Yaskawa INFORM job: OK_R2_O24B(90,0)KMOK.JBI

/JOB
//NAME OK_R2_O24B(90,0)KMOK
///FOLDERNAME X4
//POS
///NPOS 232,232,232,13,0,0
///TOOL 0
///POSTYPE PULSE
///PULSE
C00000=-110421,-114568,-128442,-17543,109310,40994
C00001=-110421,-114568,-128442,-17543,109310,40994
C00002=-114535,-118016,-126260,-17193,105500,40103
C00003=-116189,-118926,-125238,-17079,104117,39719
C00004=-122470,-118801,-125267,-16970,102934,37675
C00005=-122542,-119768,-123081,-16831,101153,37902
C00006=-122470,-118801,-125267,-16970,102934,37675
C00007=-116189,-118926,-125238,-17079,104117,39719
C00008=-115768,-121709,-122546,-16840,101244,40278
C00009=-119833,-121860,-122638,-16796,100405,38960
C00010=-115768,-121709,-122546,-16840,101244,40278
C00011=-116189,-118926,-125238,-17079,104117,39719
C00012=-114535,-118016,-126260,-17193,105500,40103
C00013=-110421,-114568,-128442,-17543,109310,40994
C00014=-126378,-115954,-129597,15290,109099,-41008
C00015=-122420,-119367,-127301,14983,105339,-40105
C00016=-120830,-120251,-126232,14883,103983,-39719
C00017=-114862,-120096,-125989,14784,102865,-37775
C00018=-115075,-121077,-123808,14669,101114,-38064
C00019=-114862,-120096,-125989,14784,102865,-37775
C00020=-120830,-120251,-126232,14883,103983,-39719
C00021=-121393,-120121,-122865,14745,102140,-40145
C00022=-117360,-120220,-122765,14697,101321,-38836
C00023=-121393,-120121,-122865,14745,102140,-40145
C00024=-120830,-120251,-126232,14883,103983,-39719
C00025=-122420,-119367,-127301,14983,105339,-40105
C00026=-126378,-115954,-129597,15290,109099,-41008
C00027=-68546,-106272,-120466,15386,126682,-61056
C00028=-65872,-117617,-121364,15125,121103,-60799
C00029=-65994,-124789,-121483,14506,117628,-61338
C00030=-65994,-124776,-119887,14364,116682,-61464
C00031=-64727,-121841,-121551,15095,118908,-60654
C00032=-66354,-118147,-119193,14717,119632,-61205
C00033=-63947,-125385,-121489,15018,116968,-60618
C00034=-66354,-118147,-119193,14717,119632,-61205
C00035=-67446,-114060,-119015,14744,121753,-61346
C00036=-69995,-103128,-118158,14981,127125,-61604
C00037=-43458,-109907,-123851,22079,119459,-51827
C00038=-39582,-118676,-123782,21672,114241,-51374
C00039=-37960,-121735,-123576,21587,112243,-51139
C00040=-38039,-122241,-121246,21299,110682,-51473
C00041=-37960,-121735,-123576,21587,112243,-51139
C00042=-39439,-119560,-121458,21353,112446,-51673
C00043=-35892,-124835,-123088,21550,109947,-50789
C00044=-39439,-119560,-121458,21353,112446,-51673
C00045=-41022,-116597,-121679,21425,114395,-51908
C00046=-44803,-108153,-121807,21787,119465,-52368
C00047=-46269,-104607,-116900,14890,131588,-81597
C00048=-45575,-117487,-118566,13929,126044,-82146
C00049=-45272,-122474,-119074,13631,123805,-82329
C00050=-45097,-121786,-116375,13476,122503,-82429
C00051=-45272,-122474,-119074,13631,123805,-82329
C00052=-54794,-132635,-122270,15461,117667,-84057
C00053=-51488,-139835,-124335,16145,114686,-83176
C00054=-54794,-132635,-122270,15461,117667,-84057
C00055=-54354,-108181,-111858,18613,130239,-82011
C00056=-56948,-114588,-113873,16794,128830,-83498
C00057=-54354,-108181,-111858,18613,130239,-82011
C00058=-54354,-108181,-111858,18613,105079,-82011
C00059=-125473,-127815,-125744,-20402,114696,66128
C00060=-144354,-128645,-122856,-20089,112993,66444
C00061=-144356,-128558,-121667,-19978,112345,66561
C00062=-143692,-123642,-120175,-20108,114021,66516
C00063=-144449,-128577,-122916,-20120,113038,66399
C00064=-144368,-128510,-121483,-19685,112887,66475
C00065=-144076,-129076,-121363,-22700,108650,60338
C00066=-144065,-129172,-121967,-22849,108765,60054
C00067=-145562,-127750,-121174,10660,122518,78224
C00068=-145562,-127687,-120572,10615,122186,78189
C00069=-144870,-122921,-119115,11103,123620,78631
C00070=-145668,-127710,-121822,10673,122944,78224
C00071=-145551,-127683,-120865,10446,122273,78190
C00072=-145550,-127738,-121466,10490,122609,78224
C00073=-145528,-127702,-122047,10145,122795,78223
C00074=-145466,-127681,-122511,8080,122804,78067
C00075=-145466,-127654,-121910,8044,122451,78039
C00076=-144776,-122735,-120395,8485,123961,78447
C00077=-145489,-127675,-123160,8112,123205,78089
C00078=-145462,-127615,-121976,8108,122518,78051
C00079=-145461,-127639,-122576,8144,122872,78079
C00080=-145470,-127509,-122616,9202,123100,78187
C00081=-145470,-127489,-122014,9161,122745,78155
C00082=-144781,-122556,-120500,9628,124248,78581
C00083=-145526,-127464,-123250,9229,123515,78201
C00084=-145457,-127452,-122138,8905,122802,78142
C00085=-145457,-127468,-122738,8946,123159,78173
C00086=-145419,-127422,-123013,7792,123191,78085
C00087=-145369,-127281,-122655,6352,123642,78005
C00088=-145369,-127269,-122086,6324,123301,77983
C00089=-144684,-122332,-120516,6740,124807,78367
C00090=-145346,-127303,-123341,6395,124049,78040
C00091=-145359,-127218,-122002,6175,123337,77977
C00092=-145359,-127231,-122569,6203,123677,77998
C00093=-145369,-127141,-122578,7278,123283,78064
C00094=-145369,-127129,-121996,7245,122933,78039
C00095=-144683,-122199,-120454,7674,124442,78435
C00096=-145369,-127140,-123243,7317,123689,78093
C00097=-145374,-127101,-121995,7642,122781,78062
C00098=-145373,-127113,-122583,7677,123134,78088
C00099=-145323,-127035,-122273,5816,123755,77984
C00100=-145301,-126904,-121478,4974,124764,77984
C00101=-145245,-126972,-122476,3510,122733,77759
C00102=-145245,-126962,-121900,3495,122385,77747
C00103=-144566,-122041,-120337,3835,123918,78081
C00104=-145130,-127078,-123177,3572,123105,77819
C00105=-145235,-126936,-121864,3341,122099,77723
C00106=-145235,-126947,-122445,3356,122451,77734
C00107=-145235,-126704,-121159,4007,122972,77833
C00108=-145235,-126667,-120590,3990,122642,77820
C00109=-144560,-121896,-119039,4346,124100,78159
C00110=-145144,-126819,-121880,4063,123351,77885
C00111=-145222,-126734,-121009,3552,122070,77754
C00112=-143543,-128240,-121764,3717,120897,78337
C00113=-144110,-127812,-122791,3542,121772,78139
C00114=-145205,-126597,-125313,3216,123991,77765
C00115=-78497,-119087,-126940,-8466,133839,13526
C00116=-78488,-120793,-123596,-8031,130934,13800
C00117=-78485,-121192,-122172,-7887,129863,13894
C00118=-78455,-120845,-123307,-7986,130735,13833
C00119=-77443,-125885,-123641,-7190,128464,14473
C00120=-78479,-121212,-122221,-7886,129884,13896
C00121=-78482,-120810,-123644,-8031,130956,13801
C00122=-78491,-119095,-126985,-8467,133863,13526
C00123=-78416,-117369,-129459,12992,98157,11559
C00124=-78415,-119818,-126610,12888,95218,11250
C00125=-78415,-120492,-125378,12858,94139,11138
C00126=-77369,-125600,-126977,12690,92378,11308
C00127=-78323,-119762,-126393,12873,95102,11269
C00128=-78420,-120510,-125276,12857,94070,11129
C00129=-78420,-119847,-126511,12886,95145,11241
C00130=-78422,-117430,-129370,12989,98073,11548
C00131=-84214,-85469,-118328,4842,91147,7442
C00132=-74059,-12147,-76922,1404,102997,10572
C00133=-133925,-71820,-61688,-34619,64887,29675
C00134=-146663,-27707,-36323,-28508,66625,23960
C00135=-151246,10085,-12654,-25869,69264,21358
C00136=-177412,39753,198,-10194,88087,11090
C00137=-178299,46865,9603,8268,86130,11567
C00138=-176438,52797,17986,7782,83863,12031
C00139=-176438,52484,19424,7790,82827,11968
C00140=-176438,52797,17986,7782,83863,12031
C00141=-176227,55662,21169,7731,83361,12069
C00142=-176438,52797,17986,7782,83863,12031
C00143=-178195,43565,7177,-9991,85692,11029
C00144=-179304,50598,16552,-9714,83440,10842
C00145=-179945,54564,20926,-9550,82718,10686
C00146=-179817,54163,20479,-9581,82800,10721
C00147=-179817,53892,21980,-9596,81755,10803
C00148=-179304,50598,16552,-9714,83440,10842
C00149=-179304,50598,16552,-9714,83440,10842
C00150=-178927,45721,9401,-9794,85349,10816
C00151=-178167,41839,2311,-9989,87773,10872
C00152=-183075,42459,3197,-17469,92450,20343
C00153=-184391,45146,9017,-17153,90080,20237
C00154=-187277,51257,17514,-16512,87509,19616
C00155=-187277,51016,18753,-16517,86658,19730
C00156=-187277,51257,17514,-16512,87509,19616
C00157=-187989,53981,20519,-16358,86938,19449
C00158=-187277,51257,17514,-16512,87509,19616
C00159=-185546,45393,8874,-16907,90057,19851
C00160=-188954,54144,18535,-20814,94698,27736
C00161=-189948,54829,23502,-24427,90749,27662
C00162=-189948,54721,24380,-24417,90207,27773
C00163=-189948,54829,23502,-24427,90749,27662
C00164=-190693,55997,24806,-24308,90350,27474
C00165=-189948,54829,23502,-24427,90749,27662
C00166=-191226,46719,10370,-23503,99774,32576
C00167=-194241,47366,13370,-23088,97565,31938
C00168=-194241,47163,14282,-23044,96951,32058
C00169=-194241,47366,13370,-23088,97565,31938
C00170=-195479,48868,14996,-22944,97022,31602
C00171=-194241,47366,13370,-23088,97565,31938
C00172=-191615,46469,10340,-23456,99568,32478
C00173=-181855,44977,8339,-27183,101400,42897
C00174=-186261,52191,18476,-27626,103380,47450
C00175=-186261,52000,19461,-27536,102751,47603
C00176=-186261,52191,18476,-27626,103380,47450
C00177=-187017,51834,18080,-27612,103190,47211
C00178=-186261,52191,18476,-27626,103380,47450
C00179=-171257,48190,12361,-32854,103470,53443
C00180=-172498,42405,8067,-32730,102732,53174
C00181=-172498,42136,9154,-32614,102046,53379
C00182=-172498,42405,8067,-32730,102732,53174
C00183=-173166,39976,5518,-32734,102755,52903
C00184=-172498,42405,8067,-32730,102732,53174
C00185=-171464,48985,12939,-32850,103438,53371
C00186=-169687,51444,12946,-33160,105162,53551
C00187=-184933,42158,3162,-30363,102223,10869
C00188=-186478,44106,8144,-29956,99900,10911
C00189=-188964,49864,16491,-29066,96066,9719
C00190=-187085,45252,9276,-29882,99600,10761
C00191=-186375,44289,9504,-29889,99288,11112
C00192=-188932,49894,16522,-29069,96073,9729
C00193=-187598,64926,30953,-23001,93658,11625
C00194=-184091,69419,36163,-18103,87388,9711
C00195=-183329,49111,13525,-21934,85838,-1831
C00196=-182560,45031,6210,-22112,88271,-2010
C00197=-164611,45054,6259,-27542,116257,62631
C00198=-165962,40795,4672,-27363,114755,62481
C00199=-168804,37690,3528,-27392,113071,61778
C00200=-167727,42077,8101,-27182,112908,62250
C00201=-168804,38233,1799,-27701,114270,61464
C00202=-172036,45397,11586,-27411,111162,60980
C00203=-173961,50198,16751,-27391,109920,60533
C00204=-173988,50269,16828,-27390,109902,60527
C00205=-175518,40442,6505,-27349,101254,50892
C00206=-176418,41479,8497,-27978,96504,46634
C00207=-174286,53569,18433,-27340,100959,51234
C00208=-172614,55478,17651,-27620,102791,51416
C00209=-179054,42000,3002,-22996,89562,-1047
C00210=-179906,45884,10050,-22784,87172,-886
C00211=-179980,55307,22142,-22805,84750,-451
C00212=-180237,47802,12025,-22705,86872,-945
C00213=-179743,45860,11189,-22831,86556,-712
C00214=-179765,55798,22804,-22861,84662,-356
C00215=-179423,51484,18060,-14503,78815,-9583
C00216=-178933,49946,16450,-4188,75758,-19147
C00217=-177518,54886,19966,-905,79614,-18236
C00218=-175510,52869,17962,2143,79991,-17090
C00219=-179383,44561,8630,-4008,77771,-19367
C00220=-179878,42216,-2358,-3772,83293,-19698
C00221=-181279,19301,-18084,-30673,107641,36259
C00222=-186954,17040,-16309,-29931,103762,35153
C00223=-186474,43263,7155,-30055,116560,25020
C00224=-185760,43661,8832,-29744,116081,25463
C00225=-186986,17160,-16198,-29927,103745,35146
C00226=-192293,22649,-14002,-21464,99552,35428
C00227=-191916,35450,-1506,-21432,98603,35730
C00228=-192278,42179,5472,-18084,93007,29470
C00229=-192157,46216,9774,-15899,90290,26168
C00230=-185951,26886,-15636,-17349,96949,27318
C00231=-180469,24600,-14591,-31088,105394,11680
BC00000=365735,697660,1075175
BC00001=365735,826919,1075175
BC00002=365735,826919,1075175
BC00003=365735,826919,1075175
BC00004=365735,826919,1075175
BC00005=365735,826919,1075175
BC00006=365735,826919,1075175
BC00007=365735,826919,1075175
BC00008=365735,826919,1075175
BC00009=365735,826919,1075175
BC00010=365735,826919,1075175
BC00011=365735,826919,1075175
BC00012=365735,826919,1075175
BC00013=365735,826919,1075175
BC00014=303667,828438,1075175
BC00015=303667,828438,1075175
BC00016=303667,828438,1075175
BC00017=303667,828438,1075175
BC00018=303667,828438,1075175
BC00019=303667,828438,1075175
BC00020=303667,828438,1075175
BC00021=303667,828438,1075175
BC00022=303667,828438,1075175
BC00023=303667,828438,1075175
BC00024=303667,828438,1075175
BC00025=303667,828438,1075175
BC00026=303667,828438,1075175
BC00027=337741,890424,1075175
BC00028=337741,890424,1075175
BC00029=337741,890424,1075175
BC00030=337741,890424,1075175
BC00031=337741,890424,1075175
BC00032=337741,890424,1075175
BC00033=337741,890424,1075175
BC00034=337741,890424,1075175
BC00035=337741,890424,1075175
BC00036=337741,890424,1075175
BC00037=224426,912763,1075175
BC00038=224426,912763,1075175
BC00039=224426,912763,1075175
BC00040=224426,912763,1075175
BC00041=224426,912763,1075175
BC00042=224426,912763,1075175
BC00043=224426,912763,1075175
BC00044=224426,912763,1075175
BC00045=224426,912763,1075175
BC00046=224426,912763,1075175
BC00047=171301,903205,1075175
BC00048=171301,903205,1075175
BC00049=171301,903205,1075175
BC00050=171301,903205,1075175
BC00051=171301,903205,1075175
BC00052=171301,903205,1075175
BC00053=171301,903205,1075175
BC00054=171301,903205,1075175
BC00055=171301,903205,1075175
BC00056=171301,903205,1075175
BC00057=171301,903205,1075175
BC00058=171301,903205,1075175
BC00059=269606,880492,1075175
BC00060=267821,875290,1075175
BC00061=267108,873210,1075175
BC00062=267108,873210,1075175
BC00063=267108,873210,1075175
BC00064=264556,874058,1075175
BC00065=269924,868703,1075175
BC00066=270646,869481,1075175
BC00067=229357,874448,1075175
BC00068=229412,873357,1075175
BC00069=229412,873357,1075175
BC00070=229412,873357,1075175
BC00071=236091,873318,1075175
BC00072=236043,874407,1075175
BC00073=249309,874312,1075175
BC00074=258931,874853,1075175
BC00075=258932,873778,1075175
BC00076=258932,873778,1075175
BC00077=258932,873778,1075175
BC00078=265217,873784,1075175
BC00079=265214,874859,1075175
BC00080=282651,874653,1075175
BC00081=282689,873584,1075175
BC00082=282689,873584,1075175
BC00083=282689,873584,1075175
BC00084=289464,873670,1075175
BC00085=289435,874740,1075175
BC00086=298152,875065,1075175
BC00087=312070,876808,1075175
BC00088=312063,875684,1075175
BC00089=312063,875684,1075175
BC00090=312063,875684,1075175
BC00091=318618,875875,1075175
BC00092=318629,877004,1075175
BC00093=336326,875802,1075175
BC00094=336344,874702,1075175
BC00095=336344,874702,1075175
BC00096=336344,874702,1075175
BC00097=342221,874261,1075175
BC00098=342191,875351,1075175
BC00099=344956,877512,1075175
BC00100=345746,880197,1075175
BC00101=367558,876774,1075175
BC00102=367507,875664,1075175
BC00103=367507,875664,1075175
BC00104=367507,875664,1075175
BC00105=374249,875310,1075175
BC00106=374309,876411,1075175
BC00107=391669,878109,1075175
BC00108=391646,876972,1075175
BC00109=391646,876972,1075175
BC00110=391646,876972,1075175
BC00111=394320,875907,1075175
BC00112=398174,874845,1075175
BC00113=398174,876946,1075175
BC00114=397796,882197,1075175
BC00115=322205,870699,1075175
BC00116=319350,870698,1075175
BC00117=318208,870697,1075175
BC00118=318208,870697,1075175
BC00119=318208,870697,1075175
BC00120=313667,870683,1075175
BC00121=314809,870684,1075175
BC00122=317664,870685,1075175
BC00123=260517,820620,1075175
BC00124=262870,823684,1075175
BC00125=263812,824910,1075175
BC00126=263812,824910,1075175
BC00127=263812,824910,1075175
BC00128=267687,824922,1075175
BC00129=266745,823696,1075175
BC00130=264392,820632,1075175
BC00131=264392,769677,1075175
BC00132=221812,674137,1075175
BC00133=202699,680494,271587
BC00134=202699,714122,185597
BC00135=202699,732276,139175
BC00136=202699,826035,116002
BC00137=202699,826035,116002
BC00138=202699,826035,116002
BC00139=202699,826035,116002
BC00140=202699,826035,116002
BC00141=202699,826035,116002
BC00142=202699,826035,116002
BC00143=202699,826035,116002
BC00144=202699,826035,116002
BC00145=202699,826035,116002
BC00146=202699,826035,116002
BC00147=202699,826035,116002
BC00148=202699,826035,116002
BC00149=202699,826035,116002
BC00150=202699,826035,116002
BC00151=202699,826035,116002
BC00152=214146,822500,117016
BC00153=214146,822500,117016
BC00154=214146,822501,117010
BC00155=214146,822501,117010
BC00156=214146,822501,117010
BC00157=214146,822501,117010
BC00158=214146,822501,117010
BC00159=214146,822500,117016
BC00160=227542,823667,115727
BC00161=227542,823667,115727
BC00162=227542,823667,115727
BC00163=227542,823667,115727
BC00164=227542,823667,115727
BC00165=227542,823667,115727
BC00166=236387,824437,114876
BC00167=236387,824436,114874
BC00168=236387,824436,114874
BC00169=236387,824436,114874
BC00170=236387,824436,114874
BC00171=236387,824436,114874
BC00172=236387,824437,114876
BC00173=241078,796619,103509
BC00174=241078,796619,103509
BC00175=241078,796619,103509
BC00176=241078,796619,103509
BC00177=241078,796619,103509
BC00178=241078,796619,103509
BC00179=245862,768255,91919
BC00180=245862,768255,91917
BC00181=245862,768255,91917
BC00182=245862,768255,91917
BC00183=245862,768255,91917
BC00184=245862,768255,91917
BC00185=245862,768255,91919
BC00186=245862,768255,91919
BC00187=217247,830516,95414
BC00188=217247,830516,95414
BC00189=217248,830516,95407
BC00190=217247,830516,95414
BC00191=217247,830516,95414
BC00192=217248,830516,95407
BC00193=217248,830516,95411
BC00194=217248,830516,95408
BC00195=217247,830516,95414
BC00196=217247,830516,95414
BC00197=224251,767755,101593
BC00198=224251,767755,101593
BC00199=224251,767755,101593
BC00200=224251,767755,101593
BC00201=224251,767755,101593
BC00202=224251,767755,101593
BC00203=224251,767755,101593
BC00204=224251,767755,101593
BC00205=224251,767755,101593
BC00206=224251,767755,101593
BC00207=224251,767755,101593
BC00208=224251,767755,101593
BC00209=207177,824936,95452
BC00210=207177,824936,95452
BC00211=207177,824936,95452
BC00212=207177,824936,95452
BC00213=207177,824936,95452
BC00214=207177,824936,95452
BC00215=207177,824936,95452
BC00216=207178,824936,95451
BC00217=207178,824936,95451
BC00218=207178,824936,95451
BC00219=207177,824936,95452
BC00220=207177,824936,95452
BC00221=219397,819007,95367
BC00222=219397,819007,95367
BC00223=219398,819006,95372
BC00224=219398,819006,95372
BC00225=219397,819007,95367
BC00226=219397,819007,95367
BC00227=219397,819007,95367
BC00228=219397,819007,95367
BC00229=219397,819007,95367
BC00230=219397,819007,95367
BC00231=219398,819006,95372
EC00000=798156,0
EC00001=798156,0
EC00002=798156,0
EC00003=798156,0
EC00004=798156,0
EC00005=798156,0
EC00006=798156,0
EC00007=798156,0
EC00008=798156,0
EC00009=798156,0
EC00010=798156,0
EC00011=798156,0
EC00012=798156,0
EC00013=798156,0
EC00014=798156,0
EC00015=798156,0
EC00016=798156,0
EC00017=798156,0
EC00018=798156,0
EC00019=798156,0
EC00020=798156,0
EC00021=798156,0
EC00022=798156,0
EC00023=798156,0
EC00024=798156,0
EC00025=798156,0
EC00026=798156,0
EC00027=798156,0
EC00028=798156,0
EC00029=798156,0
EC00030=798156,0
EC00031=798156,0
EC00032=798156,0
EC00033=798156,0
EC00034=798156,0
EC00035=798156,0
EC00036=798156,0
EC00037=798156,0
EC00038=798156,0
EC00039=798156,0
EC00040=798156,0
EC00041=798156,0
EC00042=798156,0
EC00043=798156,0
EC00044=798156,0
EC00045=798156,0
EC00046=798156,0
EC00047=798156,0
EC00048=798156,0
EC00049=798156,0
EC00050=798156,0
EC00051=798156,0
EC00052=798156,0
EC00053=798156,0
EC00054=798156,0
EC00055=798156,0
EC00056=798156,0
EC00057=798156,0
EC00058=798156,0
EC00059=798156,0
EC00060=798156,0
EC00061=798156,0
EC00062=798156,0
EC00063=798156,0
EC00064=798156,0
EC00065=798156,0
EC00066=798156,0
EC00067=798156,0
EC00068=798156,0
EC00069=798156,0
EC00070=798156,0
EC00071=798156,0
EC00072=798156,0
EC00073=798156,0
EC00074=798156,0
EC00075=798156,0
EC00076=798156,0
EC00077=798156,0
EC00078=798156,0
EC00079=798156,0
EC00080=798156,0
EC00081=798156,0
EC00082=798156,0
EC00083=798156,0
EC00084=798156,0
EC00085=798156,0
EC00086=798156,0
EC00087=798156,0
EC00088=798156,0
EC00089=798156,0
EC00090=798156,0
EC00091=798156,0
EC00092=798156,0
EC00093=798156,0
EC00094=798156,0
EC00095=798156,0
EC00096=798156,0
EC00097=798156,0
EC00098=798156,0
EC00099=798156,0
EC00100=798156,0
EC00101=798156,0
EC00102=798156,0
EC00103=798156,0
EC00104=798156,0
EC00105=798156,0
EC00106=798156,0
EC00107=798156,0
EC00108=798156,0
EC00109=798156,0
EC00110=798156,0
EC00111=798156,0
EC00112=798156,0
EC00113=798156,0
EC00114=798156,0
EC00115=798156,0
EC00116=798156,0
EC00117=798156,0
EC00118=798156,0
EC00119=798156,0
EC00120=798156,0
EC00121=798156,0
EC00122=798156,0
EC00123=798156,0
EC00124=798156,0
EC00125=798156,0
EC00126=798156,0
EC00127=798156,0
EC00128=798156,0
EC00129=798156,0
EC00130=798156,0
EC00131=798156,0
EC00132=798156,0
EC00133=798156,0
EC00134=798156,0
EC00135=798156,0
EC00136=798156,0
EC00137=798156,0
EC00138=798156,0
EC00139=798156,0
EC00140=798156,0
EC00141=798156,0
EC00142=798156,0
EC00143=798156,0
EC00144=798156,0
EC00145=798156,0
EC00146=798156,0
EC00147=798156,0
EC00148=798156,0
EC00149=798156,0
EC00150=798156,0
EC00151=798156,0
EC00152=798156,0
EC00153=798156,0
EC00154=798154,1
EC00155=798154,1
EC00156=798154,1
EC00157=798154,1
EC00158=798154,1
EC00159=798156,0
EC00160=798156,0
EC00161=798156,0
EC00162=798156,0
EC00163=798156,0
EC00164=798156,0
EC00165=798156,0
EC00166=798156,0
EC00167=798154,0
EC00168=798154,0
EC00169=798154,0
EC00170=798154,0
EC00171=798154,0
EC00172=798156,0
EC00173=798156,0
EC00174=798156,0
EC00175=798156,0
EC00176=798156,0
EC00177=798156,0
EC00178=798156,0
EC00179=798156,0
EC00180=798154,1
EC00181=798154,1
EC00182=798154,1
EC00183=798154,1
EC00184=798154,1
EC00185=798156,0
EC00186=798156,0
EC00187=798156,0
EC00188=798156,0
EC00189=798154,1
EC00190=798156,0
EC00191=798156,0
EC00192=798154,1
EC00193=798155,1
EC00194=798154,2
EC00195=798156,0
EC00196=798156,0
EC00197=798156,0
EC00198=798156,0
EC00199=798156,0
EC00200=798156,0
EC00201=798156,0
EC00202=798156,0
EC00203=798156,0
EC00204=798156,0
EC00205=798156,0
EC00206=798156,0
EC00207=798156,0
EC00208=798156,0
EC00209=798156,0
EC00210=798156,0
EC00211=798156,0
EC00212=798156,0
EC00213=798156,0
EC00214=798156,0
EC00215=798156,0
EC00216=798155,1
EC00217=798155,1
EC00218=798155,1
EC00219=798156,0
EC00220=798156,0
EC00221=798153,1
EC00222=798153,1
EC00223=798156,0
EC00224=798156,0
EC00225=798153,1
EC00226=798153,1
EC00227=798153,1
EC00228=798153,1
EC00229=798153,1
EC00230=798153,1
EC00231=798156,0
///POSTYPE BASE
///RECTAN
///RCONF 0,0,0,0,0,0,0,0,0,0,0,0,0,0,0,0,0,0,0,0,0,0,0,0
P00006=0.222,-3.123,-1.508,0.0000,0.0000,0.0000
P00021=-0.225,-6.128,-0.405,0.0000,0.0000,0.0000
P00022=0.222,-3.123,-1.508,0.0000,0.0000,0.0000
P00023=0.143,-0.036,0.682,0.0000,0.0000,0.0000
P00024=0.145,-0.552,1.326,0.0000,0.0000,0.0000
P00025=-2.003,0.006,0.728,0.0000,0.0000,0.0000
P00026=0.562,-0.002,-0.337,0.0000,0.0000,0.0000
P00027=-0.746,0.015,-9.096,0.0000,0.0000,0.0000
P00031=1.853,-0.001,-1.549,0.0000,0.0000,0.0000
P00032=1.957,0.503,-7.217,0.0000,0.0000,0.0000
///RCONF 0,0,0,0,1,0,0,0,0,0,0,0,0,0,0,0,0,0,0,0,0,0,0,0
P00033=-0.123,0.612,-5.012,0.0000,0.0000,0.0000
///RCONF 0,0,0,0,0,0,0,0,0,0,0,0,0,0,0,0,0,0,0,0,0,0,0,0
P00034=-0.304,0.773,-2.693,0.0000,0.0000,0.0000
P00035=2.817,0.591,-1.622,0.0000,0.0000,0.0000
//INST
///DATE 2024/10/31 13:36
///ATTR SC,RW
///GROUP1 RB1,BS1
///GROUP2 ST1
NOP
'OK_r2_O24B(90,0)
'
'brak tej czesci na razie
'Path S3723
SFTOF3D
MOVJ C00000 BC00000 VJ=100.00  +MOVJ EC00000 VJ=100.00
JUMP *LABEL
MOVJ C00001 BC00001 VJ=100.00  +MOVJ EC00001 VJ=100.00
MOVL C00002 BC00002 V=400.0  +MOVJ EC00002 VJ=100.00
SMOVL C00003 BC00003 V=100.0  +MOVJ EC00003
'BRAK DETALU
PAUSE
SMOVL C00004 BC00004 V=60.0  +MOVJ EC00004
SREFP 3 C00005 BC00005  +REFP EC00005
CALL JOB:SEARCH-R1-S13D
SET P031 P006
SFTON3D P031
SMOVL C00006 BC00006 V=60.0  +MOVJ EC00006
SMOVL C00007 BC00007 V=100.0  +MOVJ EC00007
SMOVL C00008 BC00008 V=60.0  +MOVJ EC00008
SREFP 3 C00009 BC00009  +REFP EC00009
CALL JOB:SEARCH-R1-S13D
SET P031 P006
SFTON3D P031
SMOVL C00010 BC00010 V=60.0  +MOVJ EC00010
SMOVL C00011 BC00011 V=100.0  +MOVJ EC00011
MOVL C00012 BC00012 V=400.0  +MOVJ EC00012 VJ=100.00
MOVL C00013 BC00013 V=1000.0  +MOVJ EC00013 VJ=100.00
'Path S3724
SFTOF3D
MOVJ C00014 BC00014 VJ=100.00  +MOVJ EC00014 VJ=100.00
MOVL C00015 BC00015 V=400.0  +MOVJ EC00015 VJ=100.00
SMOVL C00016 BC00016 V=100.0  +MOVJ EC00016
SMOVL C00017 BC00017 V=60.0  +MOVJ EC00017
SREFP 3 C00018 BC00018  +REFP EC00018
CALL JOB:SEARCH-R1-S13D
SET P032 P006
SFTON3D P032
SMOVL C00019 BC00019 V=60.0  +MOVJ EC00019
SMOVL C00020 BC00020 V=100.0  +MOVJ EC00020
SMOVL C00021 BC00021 V=60.0  +MOVJ EC00021
SREFP 3 C00022 BC00022  +REFP EC00022
CALL JOB:SEARCH-R1-S13D
SET P032 P006
SFTON3D P032
SMOVL C00023 BC00023 V=60.0  +MOVJ EC00023
SMOVL C00024 BC00024 V=100.0  +MOVJ EC00024
MOVL C00025 BC00025 V=400.0  +MOVJ EC00025 VJ=100.00
MOVL C00026 BC00026 V=1000.0  +MOVJ EC00026 VJ=100.00
'Path S3725
SFTOF3D
MOVJ C00027 BC00027 VJ=100.00  +MOVJ EC00027 VJ=100.00
MOVL C00028 BC00028 V=400.0  +MOVJ EC00028 VJ=100.00
SMOVL C00029 BC00029 V=60.0  +MOVJ EC00029
SREFP 3 C00030 BC00030  +REFP EC00030
CALL JOB:SEARCH-R1-S13D
SET P034 P006
SFTON3D P034
SMOVL C00031 BC00031 V=60.0  +MOVJ EC00031
SMOVL C00032 BC00032 V=60.0  +MOVJ EC00032
SREFP 3 C00033 BC00033  +REFP EC00033
CALL JOB:SEARCH-R1-S13D
SET P034 P006
SFTON3D P034
SMOVL C00034 BC00034 V=60.0  +MOVJ EC00034
MOVL C00035 BC00035 V=400.0  +MOVJ EC00035 VJ=100.00
MOVL C00036 BC00036 V=1000.0  +MOVJ EC00036 VJ=100.00
'Path S3726
SFTOF3D
MOVJ C00037 BC00037 VJ=100.00  +MOVJ EC00037 VJ=100.00
MOVL C00038 BC00038 V=400.0  +MOVJ EC00038 VJ=100.00
SMOVL C00039 BC00039 V=60.0  +MOVJ EC00039
SREFP 3 C00040 BC00040  +REFP EC00040
CALL JOB:SEARCH-R1-S13D
SET P035 P006
SFTON3D P035
SMOVL C00041 BC00041 V=60.0  +MOVJ EC00041
SMOVL C00042 BC00042 V=60.0  +MOVJ EC00042
SREFP 3 C00043 BC00043  +REFP EC00043
CALL JOB:SEARCH-R1-S13D
SET P035 P006
SFTON3D P035
SMOVL C00044 BC00044 V=60.0  +MOVJ EC00044
MOVL C00045 BC00045 V=400.0  +MOVJ EC00045 VJ=100.00
MOVL C00046 BC00046 V=1000.0  +MOVJ EC00046 VJ=100.00
'Path S3727
SFTOF3D
MOVJ C00047 BC00047 VJ=100.00  +MOVJ EC00047 VJ=100.00
MOVL C00048 BC00048 V=400.0  +MOVJ EC00048 VJ=100.00
SMOVL C00049 BC00049 V=60.0  +MOVJ EC00049
SREFP 3 C00050 BC00050  +REFP EC00050
CALL JOB:SEARCH-R1-S13D
SET P033 P006
SFTON3D P033
SMOVL C00051 BC00051 V=60.0  +MOVJ EC00051
SMOVL C00052 BC00052 V=60.0  +MOVJ EC00052
SREFP 3 C00053 BC00053  +REFP EC00053
CALL JOB:SEARCH-R1-S13D
SET P033 P006
SFTON3D P033
SMOVL C00054 BC00054 V=60.0  +MOVJ EC00054
SMOVL C00055 BC00055 V=60.0  +MOVJ EC00055
SREFP 3 C00056 BC00056  +REFP EC00056
CALL JOB:SEARCH-R1-S13D
SET P033 P006
SFTON3D P033
MOVJ C00057 BC00057 VJ=50.00  +MOVJ EC00057 VJ=50.00
MOVJ C00058 BC00058 VJ=50.00  +MOVJ EC00058 VJ=50.00
'Path W3728
SFTOF3D
SFTON3D P033
MOVJ C00059 BC00059 VJ=100.00  +MOVJ EC00059 VJ=100.00
SMOVL C00060 BC00060 V=400.0  +MOVJ EC00060
SMOVL C00061 BC00061 V=100.0 PL=0  +MOVJ EC00061
SREFP 1 C00062 BC00062  +REFP EC00062
SREFP 2 C00063 BC00063  +REFP EC00063
MACRO1 MJ#(0) ARGF0
ARCON
SMOVL C00064 BC00064 V=10.0  +MOVJ EC00064
SMOVL C00065 BC00065 V=10.0  +MOVJ EC00065
ARCOF
SMOVL C00066 BC00066 V=100.0  +MOVJ EC00066
SMOVL C00067 BC00067 V=100.0  +MOVJ EC00067
SMOVL C00068 BC00068 V=100.0 PL=0  +MOVJ EC00068
SREFP 1 C00069 BC00069  +REFP EC00069
SREFP 2 C00070 BC00070  +REFP EC00070
MACRO1 MJ#(0) ARGF0
ARCON
SMOVL C00071 BC00071 V=10.0  +MOVJ EC00071
ARCOF
SMOVL C00072 BC00072 V=100.0  +MOVJ EC00072
SFTON3D P035
SMOVL C00073 BC00073 V=100.0  +MOVJ EC00073
SMOVL C00074 BC00074 V=100.0  +MOVJ EC00074
SMOVL C00075 BC00075 V=100.0 PL=0  +MOVJ EC00075
SREFP 1 C00076 BC00076  +REFP EC00076
SREFP 2 C00077 BC00077  +REFP EC00077
MACRO1 MJ#(0) ARGF0
ARCON
SMOVL C00078 BC00078 V=10.0  +MOVJ EC00078
ARCOF
SMOVL C00079 BC00079 V=100.0  +MOVJ EC00079
SMOVL C00080 BC00080 V=100.0  +MOVJ EC00080
SMOVL C00081 BC00081 V=100.0 PL=0  +MOVJ EC00081
SREFP 1 C00082 BC00082  +REFP EC00082
SREFP 2 C00083 BC00083  +REFP EC00083
MACRO1 MJ#(0) ARGF0
ARCON
SMOVL C00084 BC00084 V=10.0  +MOVJ EC00084
ARCOF
SMOVL C00085 BC00085 V=100.0  +MOVJ EC00085
SMOVL C00086 BC00086 V=100.0  +MOVJ EC00086
SMOVL C00087 BC00087 V=100.0  +MOVJ EC00087
SMOVL C00088 BC00088 V=100.0 PL=0  +MOVJ EC00088
SREFP 1 C00089 BC00089  +REFP EC00089
SREFP 2 C00090 BC00090  +REFP EC00090
MACRO1 MJ#(0) ARGF0
ARCON
SMOVL C00091 BC00091 V=10.0  +MOVJ EC00091
ARCOF
SMOVL C00092 BC00092 V=100.0  +MOVJ EC00092
SMOVL C00093 BC00093 V=100.0  +MOVJ EC00093
SMOVL C00094 BC00094 V=100.0 PL=0  +MOVJ EC00094
SREFP 1 C00095 BC00095  +REFP EC00095
SREFP 2 C00096 BC00096  +REFP EC00096
MACRO1 MJ#(0) ARGF0
ARCON
SMOVL C00097 BC00097 V=10.0  +MOVJ EC00097
ARCOF
SMOVL C00098 BC00098 V=100.0  +MOVJ EC00098
SMOVL C00099 BC00099 V=100.0  +MOVJ EC00099
SMOVL C00100 BC00100 V=100.0  +MOVJ EC00100
SFTON3D P034
SMOVL C00101 BC00101 V=100.0  +MOVJ EC00101
SMOVL C00102 BC00102 V=100.0 PL=0  +MOVJ EC00102
SREFP 1 C00103 BC00103  +REFP EC00103
SREFP 2 C00104 BC00104  +REFP EC00104
MACRO1 MJ#(0) ARGF0
ARCON
SMOVL C00105 BC00105 V=10.0  +MOVJ EC00105
ARCOF
SMOVL C00106 BC00106 V=100.0  +MOVJ EC00106
SMOVL C00107 BC00107 V=100.0  +MOVJ EC00107
SMOVL C00108 BC00108 V=100.0 PL=0  +MOVJ EC00108
SREFP 1 C00109 BC00109  +REFP EC00109
SREFP 2 C00110 BC00110  +REFP EC00110
MACRO1 MJ#(0) ARGF0
ARCON
SMOVL C00111 BC00111 V=10.0  +MOVJ EC00111
SMOVL C00112 BC00112 V=10.0  +MOVJ EC00112
ARCOF
SMOVL C00113 BC00113 V=400.0  +MOVJ EC00113
SMOVL C00114 BC00114 V=1000.0  +MOVJ EC00114
SFTOF3D
'Path W3729
SFTOF3D
SFTON3D P031
MOVJ C00115 BC00115 VJ=100.00  +MOVJ EC00115 VJ=100.00
SMOVL C00116 BC00116 V=400.0  +MOVJ EC00116
SMOVL C00117 BC00117 V=100.0 PL=0  +MOVJ EC00117
SREFP 1 C00118 BC00118  +REFP EC00118
SREFP 2 C00119 BC00119  +REFP EC00119
MACRO1 MJ#(0) ARGF0
ARCON
SMOVL C00120 BC00120 V=10.0  +MOVJ EC00120
ARCOF
SMOVL C00121 BC00121 V=400.0  +MOVJ EC00121
SMOVL C00122 BC00122 V=1000.0  +MOVJ EC00122
SFTOF3D
'Path W3730
SFTOF3D
SFTON3D P032
MOVJ C00123 BC00123 VJ=100.00  +MOVJ EC00123 VJ=100.00
SMOVL C00124 BC00124 V=400.0  +MOVJ EC00124
SMOVL C00125 BC00125 V=100.0 PL=0  +MOVJ EC00125
SREFP 1 C00126 BC00126  +REFP EC00126
SREFP 2 C00127 BC00127  +REFP EC00127
MACRO1 MJ#(0) ARGF0
ARCON
SMOVL C00128 BC00128 V=10.0  +MOVJ EC00128
ARCOF
SMOVL C00129 BC00129 V=400.0  +MOVJ EC00129
SMOVL C00130 BC00130 V=1000.0  +MOVJ EC00130
SFTOF3D
MOVJ C00131 BC00131 VJ=100.00  +MOVJ EC00131 VJ=100.00
MOVJ C00132 BC00132 VJ=100.00  +MOVJ EC00132 VJ=100.00
'dotad odkoment
'down
*LABEL
MOVJ C00133 BC00133 VJ=100.00  +MOVJ EC00133 VJ=100.00
MOVJ C00134 BC00134 VJ=100.00  +MOVJ EC00134 VJ=100.00
MOVJ C00135 BC00135 VJ=15.00  +MOVJ EC00135 VJ=100.00
'Path S3731
SFTOF3D
MOVJ C00136 BC00136 VJ=30.00  +MOVJ EC00136 VJ=100.00
MOVJ C00137 BC00137 VJ=30.00  +MOVJ EC00137 VJ=0.78
SMOVL C00138 BC00138 V=166.7  +MOVJ EC00138
SREFP 3 C00139 BC00139  +REFP EC00139
CALL JOB:SEARCH-R1-S13D
SET P025 P006
SFTON3D P025
SMOVL C00140 BC00140 V=100.0  +MOVJ EC00140
SREFP 3 C00141 BC00141  +REFP EC00141
CALL JOB:SEARCH-R1-S13D
SET P025 P006
SFTON3D P025
SMOVL C00142 BC00142 V=250.0  +MOVJ EC00142
SFTOF3D
MOVL C00143 BC00143 V=400.0  +MOVJ EC00143 VJ=100.00
SMOVL C00144 BC00144 V=100.0  +MOVJ EC00144
SREFP 3 C00145 BC00145  +REFP EC00145
CALL JOB:SEARCH-R1-S13D
SET P021 P006
SFTON3D P021
SMOVL C00146 BC00146 V=83.3  +MOVJ EC00146
SREFP 3 C00147 BC00147  +REFP EC00147
CALL JOB:SEARCH-R1-S13D
SET P021 P006
SFTON3D P021
SMOVL C00148 BC00148 V=100.0  +MOVJ EC00148
SMOVL C00149 BC00149 V=100.0  +MOVJ EC00149
MOVL C00150 BC00150 V=400.0  +MOVJ EC00150 VJ=100.00
MOVL C00151 BC00151 V=1000.0  +MOVJ EC00151 VJ=100.00
'Path S3732
SFTOF3D
MOVJ C00152 BC00152 VJ=100.00  +MOVJ EC00152 VJ=100.00
MOVL C00153 BC00153 V=400.0  +MOVJ EC00153 VJ=100.00
SMOVL C00154 BC00154 V=100.0  +MOVJ EC00154
SREFP 3 C00155 BC00155  +REFP EC00155
CALL JOB:SEARCH-R1-S13D
SET P022 P006
SFTON3D P022
SMOVL C00156 BC00156 V=100.0  +MOVJ EC00156
SREFP 3 C00157 BC00157  +REFP EC00157
CALL JOB:SEARCH-R1-S13D
SET P022 P006
SFTON3D P022
SMOVL C00158 BC00158 V=100.0  +MOVJ EC00158
SFTOF3D
MOVL C00159 BC00159 V=400.0  +MOVJ EC00159 VJ=100.00
MOVL C00160 BC00160 V=500.0  +MOVJ EC00160 VJ=100.00
SMOVL C00161 BC00161 V=166.7  +MOVJ EC00161
SREFP 3 C00162 BC00162  +REFP EC00162
CALL JOB:SEARCH-R1-S13D
SET P027 P006
SFTON3D P027
SMOVL C00163 BC00163 V=100.0  +MOVJ EC00163
SREFP 3 C00164 BC00164  +REFP EC00164
CALL JOB:SEARCH-R1-S13D
SET P027 P006
SFTON3D P027
SMOVL C00165 BC00165 V=166.7  +MOVJ EC00165
'Path S3733
SFTOF3D
MOVL C00166 BC00166 V=400.0  +MOVJ EC00166 VJ=100.00
SMOVL C00167 BC00167 V=166.7  +MOVJ EC00167
SREFP 3 C00168 BC00168  +REFP EC00168
CALL JOB:SEARCH-R1-S13D
SET P023 P006
SFTON3D P023
SMOVL C00169 BC00169 V=100.0  +MOVJ EC00169
SREFP 3 C00170 BC00170  +REFP EC00170
CALL JOB:SEARCH-R1-S13D
SET P023 P006
SFTON3D P023
SMOVL C00171 BC00171 V=166.7  +MOVJ EC00171
MOVL C00172 BC00172 V=400.0  +MOVJ EC00172 VJ=100.00
'Path S3734
SFTOF3D
MOVJ C00173 BC00173 VJ=50.00  +MOVJ EC00173 VJ=50.00
SMOVL C00174 BC00174 V=166.7  +MOVJ EC00174
SREFP 3 C00175 BC00175  +REFP EC00175
CALL JOB:SEARCH-R1-S13D
SET P026 P006
SFTON3D P026
SMOVL C00176 BC00176 V=166.7  +MOVJ EC00176
SREFP 3 C00177 BC00177  +REFP EC00177
CALL JOB:SEARCH-R1-S13D
SET P026 P006
SFTON3D P026
SMOVL C00178 BC00178 V=166.7  +MOVJ EC00178
MOVL C00179 BC00179 V=400.0  +MOVJ EC00179 VJ=100.00
SMOVL C00180 BC00180 V=100.0  +MOVJ EC00180
SREFP 3 C00181 BC00181  +REFP EC00181
CALL JOB:SEARCH-R1-S13D
SET P024 P006
SFTON3D P024
SMOVL C00182 BC00182 V=100.0  +MOVJ EC00182
SREFP 3 C00183 BC00183  +REFP EC00183
CALL JOB:SEARCH-R1-S13D
SET P024 P006
SFTON3D P024
SMOVL C00184 BC00184 V=100.0  +MOVJ EC00184
MOVL C00185 BC00185 V=400.0  +MOVJ EC00185 VJ=100.00
MOVL C00186 BC00186 V=1000.0  +MOVJ EC00186 VJ=100.00
'Path W3735
SFTOF3D
MOVJ C00187 BC00187 VJ=100.00  +MOVJ EC00187 VJ=100.00
SMOVL C00188 BC00188 V=400.0  +MOVJ EC00188
SFTON3D P027
SMOVL C00189 BC00189 V=166.7 PL=0  +MOVJ EC00189
SREFP 1 C00190 BC00190  +REFP EC00190
SREFP 2 C00191 BC00191  +REFP EC00191
MACRO1 MJ#(0) ARGF21
ARCON
SWVON WEV#(100)
SMOVC C00192 BC00192 V=8.3  +MOVJ EC00192
SFTON3D P022
SMOVC C00193 BC00193 V=8.3  +MOVJ EC00193
SFTON3D P021
SMOVC C00194 BC00194 V=8.3  +MOVJ EC00194
ARCOF
SWVOF
SMOVL C00195 BC00195 V=400.0  +MOVJ EC00195
SMOVL C00196 BC00196 V=1000.0  +MOVJ EC00196
SFTOF3D
'Path W3737
SFTOF3D
SFTON3D P024
MOVJ C00197 BC00197 VJ=100.00  +MOVJ EC00197 VJ=100.00
SMOVL C00198 BC00198 V=400.0  +MOVJ EC00198
SMOVL C00199 BC00199 V=166.7 PL=0  +MOVJ EC00199
SREFP 1 C00200 BC00200  +REFP EC00200
SREFP 2 C00201 BC00201  +REFP EC00201
MACRO1 MJ#(0) ARGF21
ARCON
SWVON WEV#(100)
SMOVL C00202 BC00202 V=8.3  +MOVJ EC00202
SMOVL C00203 BC00203 V=8.3  +MOVJ EC00203
SMOVC C00204 BC00204 V=8.3  +MOVJ EC00204
SFTON3D P026
SMOVC C00205 BC00205 V=8.3  +MOVJ EC00205
SMOVC C00206 BC00206 V=8.3  +MOVJ EC00206
ARCOF
SWVOF
SMOVL C00207 BC00207 V=400.0  +MOVJ EC00207
SMOVL C00208 BC00208 V=1000.0  +MOVJ EC00208
SFTOF3D
'Path W3736
SFTOF3D
SFTON3D P021
MOVJ C00209 BC00209 VJ=100.00  +MOVJ EC00209 VJ=100.00
SMOVL C00210 BC00210 V=400.0  +MOVJ EC00210
SFTON3D P021
SMOVL C00211 BC00211 V=166.7 PL=0  +MOVJ EC00211
SREFP 1 C00212 BC00212  +REFP EC00212
SREFP 2 C00213 BC00213  +REFP EC00213
MACRO1 MJ#(0) ARGF21
ARCON
SWVON WEV#(100)
SMOVC C00214 BC00214 V=8.3  +MOVJ EC00214
SMOVC C00215 BC00215 V=8.3  +MOVJ EC00215
SFTON3D P025
SMOVC C00216 BC00216 V=8.3  +MOVJ EC00216
SMOVC C00217 BC00217 V=8.3  +MOVJ EC00217
SMOVL C00218 BC00218 V=8.3  +MOVJ EC00218
ARCOF
SWVOF
SFTOF3D
SMOVL C00219 BC00219 V=400.0  +MOVJ EC00219
SMOVL C00220 BC00220 V=1000.0  +MOVJ EC00220
SFTOF3D
'Path W3738
SFTOF3D
SFTON3D P026
SMOVL C00221 BC00221 V=583.3  +MOVJ EC00221
SMOVL C00222 BC00222 V=166.7 PL=0  +MOVJ EC00222
SREFP 1 C00223 BC00223  +REFP EC00223
SREFP 2 C00224 BC00224  +REFP EC00224
MACRO1 MJ#(0) ARGF21
ARCON
SWVON WEV#(100)
SMOVC C00225 BC00225 V=8.3  +MOVJ EC00225
SMOVC C00226 BC00226 V=8.3  +MOVJ EC00226
SFTON3D P023
SMOVC C00227 BC00227 V=8.3  +MOVJ EC00227
SFTON3D P027
SMOVC C00228 BC00228 V=8.3  +MOVJ EC00228
SMOVC C00229 BC00229 V=8.3  +MOVJ EC00229
ARCOF
SWVOF
SFTOF3D
SMOVL C00230 BC00230 V=400.0  +MOVJ EC00230
SMOVL C00231 BC00231 V=1000.0  +MOVJ EC00231
SFTOF3D
END
